// TIA Portal V19 export
DATA_BLOCK "Dispenser_Main_DB"   // DB4
// stored: InstanceOfName Dispenser_Main, InstanceOfType FB
"Dispenser_Main"
BEGIN
END_DATA_BLOCK
